INTERFACE I_Conexion

METHOD EstablecerConexion : BOOL
VAR_INPUT
END_VAR
END_METHOD

END_INTERFACE

(* stored: Version 1.1.0.1, ProductVersion 3.1.4024.12
   Itf I_Conexion: Id {768cbc09-99c5-4675-a36b-5351285e5ae5}
   Method EstablecerConexion: Id {778a6dc2-3cc8-4763-99cf-3cef36abdc49} *)
